TYPE DATA :
UNION
stTest : STRING;
  arTest : ARRAY[0..79] OF BYTE;
END_UNION
END_TYPE

(* stored: Version 1.1.0.1
   DUT DATA: Id {c603f045-6ee1-49a5-addd-ba03e2a4bd67} *)
